(* IEC 61131-3 sources: AXOpen/src/integrations/ctrl/src/Examples/ix-core-IxObject, 1 file *)

(* ---- IxObjectExample.st ---- *)
USING AXOpen.Core;

NAMESPACE IxObjectExamples
//<IxContext>
    CLASS PUBLIC MyContext EXTENDS  AXOpen.Core.IxContext
        VAR
            _myObject : IxObject;
        END_VAR
        METHOD PROTECTED OVERRIDE Main
            _myObject.Initialize(THIS);
        END_METHOD
    END_CLASS
//</IxContext>
//<IxObject>
    CLASS PUBLIC MyParentObject  EXTENDS IxContext
        VAR
            _myChildObject  : IxObject;
        END_VAR
        METHOD PROTECTED OVERRIDE Main
            _myChildObject.Initialize(THIS);
        END_METHOD
    END_CLASS
//</IxObject>
END_NAMESPACE
